    // LREAL
    IF UDINT_TO_INT(Expected.TypeClass) = IBaseLibrary.TypeClass.TYPE_LREAL THEN
        MEMCPY(destAddr := ADR(lrealExpected), srcAddr := Expected.pValue, n := SIZEOF(LREAL));
        MEMCPY(destAddr := ADR(lrealActual), srcAddr := Actual.pValue, n := SIZEOF(LREAL));
        AssertEquals_LREAL(Expected := lrealExpected, Actual := lrealActual, Delta := 0.0, Message := Message);
        RETURN;
    END_IF

    // LTIME
    IF UDINT_TO_INT(Expected.TypeClass) = IBaseLibrary.TypeClass.TYPE_LTIME THEN
        MEMCPY(destAddr := ADR(ltimeExpected), srcAddr := Expected.pValue, n := SIZEOF(LTIME));
        MEMCPY(destAddr := ADR(ltimeActual), srcAddr := Actual.pValue, n := SIZEOF(LTIME));
        AssertEquals_LTIME(Expected := ltimeExpected, Actual := ltimeActual, Message := Message);
        RETURN;
    END_IF

    // LWORD
    IF UDINT_TO_INT(Expected.TypeClass) = IBaseLibrary.TypeClass.TYPE_LWORD THEN
        MEMCPY(destAddr := ADR(lwordExpected), srcAddr := Expected.pValue, n := SIZEOF(LWORD));
        MEMCPY(destAddr := ADR(lwordActual), srcAddr := Actual.pValue, n := SIZEOF(LWORD));
        AssertEquals_LWORD(Expected := lwordExpected, Actual := lwordActual, Message := Message);
        RETURN;
    END_IF

    // REAL
    IF UDINT_TO_INT(Expected.TypeClass) = IBaseLibrary.TypeClass.TYPE_REAL THEN
        MEMCPY(destAddr := ADR(realExpected), srcAddr := Expected.pValue, n := SIZEOF(REAL));
        MEMCPY(destAddr := ADR(realActual), srcAddr := Actual.pValue, n := SIZEOF(REAL));
        AssertEquals_REAL(Expected := realExpected, Actual := realActual, Delta := 0.0, Message := Message);
        RETURN;
    END_IF

    // SINT
    IF UDINT_TO_INT(Expected.TypeClass) = IBaseLibrary.TypeClass.TYPE_SINT THEN
        MEMCPY(destAddr := ADR(sintExpected), srcAddr := Expected.pValue, n := SIZEOF(SINT));
        MEMCPY(destAddr := ADR(sintActual), srcAddr := Actual.pValue, n := SIZEOF(SINT));
        AssertEquals_SINT(Expected := sintExpected, Actual := sintActual, Message := Message);
        RETURN;
    END_IF

    // STRING
    IF UDINT_TO_INT(Expected.TypeClass) = IBaseLibrary.TypeClass.TYPE_STRING THEN
        MEMCPY(destAddr := ADR(stringExpected), srcAddr := Expected.pValue, n := DINT_TO_UDINT(Expected.diSize));
        MEMCPY(destAddr := ADR(stringActual), srcAddr := Actual.pValue, n := DINT_TO_UDINT(Actual.diSize));
        AssertEquals_STRING(Expected := stringExpected, Actual := stringActual, Message := Message);
        RETURN;
    END_IF

    // WSTRING
    IF UDINT_TO_INT(Expected.TypeClass) = IBaseLibrary.TypeClass.TYPE_WSTRING THEN
        MEMCPY(destAddr := ADR(wstringExpected), srcAddr := Expected.pValue, n := DINT_TO_UDINT(Expected.diSize));
        MEMCPY(destAddr := ADR(wstringActual), srcAddr := Actual.pValue, n := DINT_TO_UDINT(Actual.diSize));
        AssertEquals_WSTRING(Expected := wstringExpected, Actual := wstringActual, Message := Message);
        RETURN;
    END_IF

    // TIME
    IF UDINT_TO_INT(Expected.TypeClass) = IBaseLibrary.TypeClass.TYPE_TIME THEN
        MEMCPY(destAddr := ADR(timeExpected), srcAddr := Expected.pValue, n := SIZEOF(TIME));
        MEMCPY(destAddr := ADR(timeActual), srcAddr := Actual.pValue, n := SIZEOF(TIME));
        AssertEquals_TIME(Expected := timeExpected, Actual := timeActual, Message := Message);
        RETURN;
    END_IF

    // TIME_OF_DAY
    IF UDINT_TO_INT(Expected.TypeClass) = IBaseLibrary.TypeClass.TYPE_TIMEOFDAY THEN
        MEMCPY(destAddr := ADR(timeOfDayExpected), srcAddr := Expected.pValue, n := SIZEOF(TIME_OF_DAY));
        MEMCPY(destAddr := ADR(timeOfDayActual), srcAddr := Actual.pValue, n := SIZEOF(TIME_OF_DAY));
        AssertEquals_TIME_OF_DAY(Expected := timeOfDayExpected, Actual := timeOfDayActual, Message := Message);
        RETURN;
    END_IF

    // UDINT
    IF UDINT_TO_INT(Expected.TypeClass) = IBaseLibrary.TypeClass.TYPE_UDINT THEN
        MEMCPY(destAddr := ADR(udintExpected), srcAddr := Expected.pValue, n := SIZEOF(UDINT));
        MEMCPY(destAddr := ADR(udintActual), srcAddr := Actual.pValue, n := SIZEOF(UDINT));
        AssertEquals_UDINT(Expected := udintExpected, Actual := udintActual, Message := Message);
        RETURN;
    END_IF

    // UINT
    IF UDINT_TO_INT(Expected.TypeClass) = IBaseLibrary.TypeClass.TYPE_UINT THEN
        MEMCPY(destAddr := ADR(uintExpected), srcAddr := Expected.pValue, n := SIZEOF(UINT));
        MEMCPY(destAddr := ADR(uintActual), srcAddr := Actual.pValue, n := SIZEOF(UINT));
        AssertEquals_UINT(Expected := uintExpected, Actual := uintActual, Message := Message);
        RETURN;
    END_IF

    // ULINT
    IF UDINT_TO_INT(Expected.TypeClass) = IBaseLibrary.TypeClass.TYPE_ULINT THEN
        MEMCPY(destAddr := ADR(ulintExpected), srcAddr := Expected.pValue, n := SIZEOF(ULINT));
        MEMCPY(destAddr := ADR(ulintActual), srcAddr := Actual.pValue, n := SIZEOF(ULINT));
        AssertEquals_ULINT(Expected := ulintExpected, Actual := ulintActual, Message := Message);
        RETURN;
    END_IF

    // USINT
    IF UDINT_TO_INT(Expected.TypeClass) = IBaseLibrary.TypeClass.TYPE_USINT THEN
        MEMCPY(destAddr := ADR(usintExpected), srcAddr := Expected.pValue, n := SIZEOF(USINT));
        MEMCPY(destAddr := ADR(usintActual), srcAddr := Actual.pValue, n := SIZEOF(USINT));
        AssertEquals_USINT(Expected := usintExpected, Actual := usintActual, Message := Message);
        RETURN;
    END_IF

    // WORD
    IF UDINT_TO_INT(Expected.TypeClass) = IBaseLibrary.TypeClass.TYPE_WORD THEN
        MEMCPY(destAddr := ADR(wordExpected), srcAddr := Expected.pValue, n := SIZEOF(WORD));
        MEMCPY(destAddr := ADR(wordActual), srcAddr := Actual.pValue, n := SIZEOF(WORD));
        AssertEquals_WORD(Expected := wordExpected, Actual := wordActual, Message := Message);
        RETURN;
    END_IF

END_IF

(* If we've come to this row, it means that the data input is not any of the standard primitive data types, and thus
   we need to do special handling *)
TestInstancePath := AddTestNameToInstancePath(TestInstancePath := FindTestSuiteInstancePath());

IF DataTypesNotEquals THEN
    ExpectedDataString := CONCAT(STR1 := '(Type class = ', STR2 := F_AnyTypeClassToString((Expected.TypeClass)));
    ExpectedDataString := CONCAT(STR1 := ExpectedDataString, STR2 := ')');
    ActualDataString := CONCAT(STR1 := '(Type class = ', STR2 := F_AnyTypeClassToString(Actual.TypeClass));
    ActualDataString := CONCAT(STR1 := ActualDataString, STR2 := ')');
ELSIF DataSizeNotEquals THEN
    (* Take special care of STRING and WSTRING, as these can be declared with different sizes,
       although their content might be the same *)
    IF UDINT_TO_INT(Expected.TypeClass) = IBaseLibrary.TypeClass.TYPE_STRING THEN
        MEMCPY(destAddr := ADR(stringExpected), srcAddr := Expected.pValue, n := DINT_TO_UDINT(Expected.diSize));
        MEMCPY(destAddr := ADR(stringActual), srcAddr := Actual.pValue, n := DINT_TO_UDINT(Actual.diSize));
        ExpectedDataString := CONCAT(STR1 := '(Data size (LEN) = ', STR2 := INT_TO_STRING(LEN(STR := stringExpected)));
        ActualDataString := CONCAT(STR1 := '(Data size (LEN) = ', STR2 := INT_TO_STRING(LEN(STR := stringActual)));
    ELSIF UDINT_TO_INT(Expected.TypeClass) = IBaseLibrary.TypeClass.TYPE_WSTRING THEN
        MEMCPY(destAddr := ADR(wstringExpected), srcAddr := Expected.pValue, n := DINT_TO_UDINT(Expected.diSize));
        MEMCPY(destAddr := ADR(wstringActual), srcAddr := Actual.pValue, n := DINT_TO_UDINT(Actual.diSize));
        ExpectedDataString := CONCAT(STR1 := '(Data size (WLEN) = ', STR2 := INT_TO_STRING(WLEN(STR := wstringExpected)));
        ActualDataString := CONCAT(STR1 := '(Data size (WLEN) = ', STR2 := INT_TO_STRING(WLEN(STR := wstringActual)));
    ELSE
        ExpectedDataString := CONCAT(STR1 := '(Data size = ', STR2 := DINT_TO_STRING(Expected.diSize));
        ActualDataString := CONCAT(STR1 := '(Data size = ', STR2 := DINT_TO_STRING(Actual.diSize));
    END_IF
    ExpectedDataString := CONCAT(STR1 := ExpectedDataString, STR2 := ')');
    ActualDataString := CONCAT(STR1 := ActualDataString, STR2 := ')');
ELSIF DataContentNotEquals THEN
    FOR Count := 0 TO MIN(Expected.diSize-1, 38) BY 1 DO // One byte will equal two characters (example: 255 = 0xff, 1 = 0x01)
        ExpectedDataString := CONCAT(STR1 := ExpectedDataString,
                                                  STR2 := BYTE_TO_HEXSTR(in := Expected.pValue[Count],
                                                                                       iPrecision := 2,
                                                                                       bLoCase := FALSE));
    END_FOR
    ExpectedDataString := CONCAT(STR1 := '0x', STR2 := ExpectedDataString);

    FOR Count := 0 TO MIN(Actual.diSize-1, 38) BY 1 DO // One byte will equal two characters (example: 255 = 0xff, 1 = 0x01)
        ActualDataString := CONCAT(STR1 := ActualDataString,
                                                STR2 := BYTE_TO_HEXSTR(in := Actual.pValue[Count],
                                                                                     iPrecision := 2,
                                                                                     bLoCase := FALSE));
    END_FOR
    ActualDataString := CONCAT(STR1 := '0x', STR2 := ActualDataString);
END_IF

AssertResults.ReportResult(ExpectedSize := DINT_TO_UDINT(Expected.diSize),
                           ExpectedTypeClass := UDINT_TO_INT(Expected.TypeClass),
                           ExpectedValue := Expected.pValue,
                           ActualSize := DINT_TO_UDINT(Actual.diSize),
                           ActualTypeClass := UDINT_TO_INT(Actual.TypeClass),
                           ActualValue := Actual.pValue,
                           Message := Message,
                           TestInstancePath := TestInstancePath,
                           AlreadyReported => AlreadyReported);

IF NOT AlreadyReported AND (DataTypesNotEquals OR DataSizeNotEquals OR DataContentNotEquals) THEN
    SetTestFailed(AssertionType := E_AssertionType.Type_ANY,
                  AssertionMessage := Message);

    AssertMessageFormatter.LogAssertFailure(Expected := ExpectedDataString,
                                            Actual := ActualDataString,
                                            Message := Message,
                                            TestInstancePath := TestInstancePath);
END_IF
END_METHOD

// Asserts that two BOOLs are equal. If they are not, an assertion error is created.
METHOD PUBLIC AssertEquals_BOOL
VAR_INPUT
    Expected : BOOL; // BOOL expected value
    Actual : BOOL; // BOOL actual value
    Message : T_MaxString; // The identifying message for the assertion error
END_VAR
VAR
    AlreadyReported : BOOL;
    TestInstancePath : T_MaxString;
END_VAR
IF GVL_TcUnit.IgnoreCurrentTest OR GVL_TcUnit.CurrentTestIsFinished THEN
    RETURN;
END_IF

TestInstancePath := AddTestNameToInstancePath(TestInstancePath := FindTestSuiteInstancePath());

AssertResults.ReportResult(ExpectedSize := SIZEOF(Expected),
                           ExpectedTypeClass := IBaseLibrary.TypeClass.TYPE_BOOL,
                           ExpectedValue := ADR(Expected),
                           ActualSize := SIZEOF(Actual),
                           ActualTypeClass := IBaseLibrary.TypeClass.TYPE_BOOL,
                           ActualValue := ADR(Actual),
                           Message := Message,
                           TestInstancePath := TestInstancePath,
                           AlreadyReported => AlreadyReported);

IF NOT AlreadyReported AND Expected <> Actual THEN
    SetTestFailed(AssertionType := E_AssertionType.Type_BOOL,
                  AssertionMessage := Message);

    AssertMessageFormatter.LogAssertFailure(Expected := BOOL_TO_STRING(Expected),
                                            Actual := BOOL_TO_STRING(Actual),
                                            Message := Message,
                                            TestInstancePath := TestInstancePath);
END_IF
END_METHOD

// Asserts that two BYTEs are equal. If they are not, an assertion error is created.
METHOD PUBLIC AssertEquals_BYTE
VAR_INPUT
    Expected : BYTE; // BYTE expected value
    Actual : BYTE; // BYTE actual value
    Message : T_MaxString; // The identifying message for the assertion error
END_VAR
VAR
    TestInstancePath : T_MaxString;
    AlreadyReported : BOOL;
END_VAR
IF GVL_TcUnit.IgnoreCurrentTest OR GVL_TcUnit.CurrentTestIsFinished THEN
    RETURN;
END_IF

TestInstancePath := AddTestNameToInstancePath(TestInstancePath := FindTestSuiteInstancePath());

AssertResults.ReportResult(ExpectedSize := SIZEOF(Expected),
                           ExpectedTypeClass := IBaseLibrary.TypeClass.TYPE_BYTE,
                           ExpectedValue := ADR(Expected),
                           ActualSize := SIZEOF(Actual),
                           ActualTypeClass := IBaseLibrary.TypeClass.TYPE_BYTE,
                           ActualValue := ADR(Actual),
                           Message := Message,
                           TestInstancePath := TestInstancePath,
                           AlreadyReported => AlreadyReported);

IF NOT AlreadyReported AND Expected <> Actual THEN
    SetTestFailed(AssertionType := E_AssertionType.Type_BYTE,
                  AssertionMessage := Message);

    AssertMessageFormatter.LogAssertFailure(Expected := CONCAT(
                                                       STR1 := '0x',
                                                       STR2 := BYTE_TO_HEXSTR(in := Expected,
                                                                                            iPrecision := 2,
                                                                                            bLoCase := FALSE)),
                                            Actual := CONCAT(
                                                       STR1 := '0x',
                                                       STR2 := BYTE_TO_HEXSTR(in := Actual,
                                                                                            iPrecision := 2,
                                                                                            bLoCase := FALSE)),
                                            Message := Message,
                                            TestInstancePath := TestInstancePath);
END_IF
END_METHOD

// Asserts that two DATEs are equal. If they are not, an assertion error is created.
METHOD PUBLIC AssertEquals_DATE
VAR_INPUT
    Expected : DATE; // DATE expected value
    Actual : DATE; // DATE actual value
    Message : T_MaxString; // The identifying message for the assertion error
END_VAR
VAR
    TestInstancePath : T_MaxString;
    AlreadyReported : BOOL;
END_VAR
IF GVL_TcUnit.IgnoreCurrentTest OR GVL_TcUnit.CurrentTestIsFinished THEN
    RETURN;
END_IF

TestInstancePath := AddTestNameToInstancePath(TestInstancePath := FindTestSuiteInstancePath());

AssertResults.ReportResult(ExpectedSize := SIZEOF(Expected),
                           ExpectedTypeClass := IBaseLibrary.TypeClass.TYPE_DATE,
                           ExpectedValue := ADR(Expected),
                           ActualSize := SIZEOF(Actual),
                           ActualTypeClass := IBaseLibrary.TypeClass.TYPE_DATE,
                           ActualValue := ADR(Actual),
                           Message := Message,
                           TestInstancePath := TestInstancePath,
                           AlreadyReported => AlreadyReported);

IF NOT AlreadyReported AND Expected <> Actual THEN
    SetTestFailed(AssertionType := E_AssertionType.Type_DATE,
                  AssertionMessage := Message);

    AssertMessageFormatter.LogAssertFailure(Expected := DATE_TO_STRING(Expected),
                                            Actual := DATE_TO_STRING(Actual),
                                            Message := Message,
                                            TestInstancePath := TestInstancePath);
END_IF
END_METHOD

// Asserts that two DATE_AND_TIMEs are equal. If they are not, an assertion error is created.
METHOD PUBLIC AssertEquals_DATE_AND_TIME
VAR_INPUT
    Expected : DATE_AND_TIME; // DATE_AND_TIME expected value
    Actual : DATE_AND_TIME; // DATE_AND_TIME actual value
    Message : T_MaxString; // The identifying message for the assertion error
END_VAR
VAR
    TestInstancePath : T_MaxString;
    AlreadyReported : BOOL;
END_VAR
IF GVL_TcUnit.IgnoreCurrentTest OR GVL_TcUnit.CurrentTestIsFinished THEN
    RETURN;
END_IF

TestInstancePath := AddTestNameToInstancePath(TestInstancePath := FindTestSuiteInstancePath());

AssertResults.ReportResult(ExpectedSize := SIZEOF(Expected),
                           ExpectedTypeClass := IBaseLibrary.TypeClass.TYPE_DATEANDTIME,
                           ExpectedValue := ADR(Expected),
                           ActualSize := SIZEOF(Actual),
                           ActualTypeClass := IBaseLibrary.TypeClass.TYPE_DATEANDTIME,
                           ActualValue := ADR(Actual),
                           Message := Message,
                           TestInstancePath := TestInstancePath,
                           AlreadyReported => AlreadyReported);

IF NOT AlreadyReported AND Expected <> Actual THEN
    SetTestFailed(AssertionType := E_AssertionType.Type_DATE_AND_TIME,
                  AssertionMessage := Message);

    AssertMessageFormatter.LogAssertFailure(Expected := DT_TO_STRING(Expected),
                                            Actual := DT_TO_STRING(Actual),
                                            Message := Message,
                                            TestInstancePath := TestInstancePath);
END_IF
END_METHOD

// Asserts that two DINTs are equal. If they are not, an assertion error is created.
METHOD PUBLIC AssertEquals_DINT
VAR_INPUT
    Expected : DINT; // DINT expected value
    Actual : DINT; // DINT actual value
    Message : T_MaxString; // The identifying message for the assertion error
END_VAR
VAR
    TestInstancePath : T_MaxString;
    AlreadyReported : BOOL;
END_VAR
IF GVL_TcUnit.IgnoreCurrentTest OR GVL_TcUnit.CurrentTestIsFinished THEN
    RETURN;
END_IF

TestInstancePath := AddTestNameToInstancePath(TestInstancePath := FindTestSuiteInstancePath());

AssertResults.ReportResult(ExpectedSize := SIZEOF(Expected),
                           ExpectedTypeClass := IBaseLibrary.TypeClass.TYPE_DINT,
                           ExpectedValue := ADR(Expected),
                           ActualSize := SIZEOF(Actual),
                           ActualTypeClass := IBaseLibrary.TypeClass.TYPE_DINT,
                           ActualValue := ADR(Actual),
                           Message := Message,
                           TestInstancePath := TestInstancePath,
                           AlreadyReported => AlreadyReported);

IF NOT AlreadyReported AND Expected <> Actual THEN
    SetTestFailed(AssertionType := E_AssertionType.Type_DINT,
                  AssertionMessage := Message);

    AssertMessageFormatter.LogAssertFailure(Expected := DINT_TO_STRING(Expected),
                                            Actual := DINT_TO_STRING(Actual),
                                            Message := Message,
                                            TestInstancePath := TestInstancePath);
END_IF
END_METHOD

// Asserts that two DWORDs are equal. If they are not, an assertion error is created.
METHOD PUBLIC AssertEquals_DWORD
VAR_INPUT
    Expected : DWORD; // DWORD expected value
    Actual : DWORD; // DWORD actual value
    Message : T_MaxString; // The identifying message for the assertion error
END_VAR
VAR
    TestInstancePath : T_MaxString;
    AlreadyReported : BOOL;
END_VAR
IF GVL_TcUnit.IgnoreCurrentTest OR GVL_TcUnit.CurrentTestIsFinished THEN
    RETURN;
END_IF

TestInstancePath := AddTestNameToInstancePath(TestInstancePath := FindTestSuiteInstancePath());

AssertResults.ReportResult(ExpectedSize := SIZEOF(Expected),
                           ExpectedTypeClass := IBaseLibrary.TypeClass.TYPE_DWORD,
                           ExpectedValue := ADR(Expected),
                           ActualSize := SIZEOF(Actual),
                           ActualTypeClass := IBaseLibrary.TypeClass.TYPE_DWORD,
                           ActualValue := ADR(Actual),
                           Message := Message,
                           TestInstancePath := TestInstancePath,
                           AlreadyReported => AlreadyReported);

IF NOT AlreadyReported AND Expected <> Actual THEN
    SetTestFailed(AssertionType := E_AssertionType.Type_DWORD,
                  AssertionMessage := Message);

    AssertMessageFormatter.LogAssertFailure(Expected := CONCAT(
                                                            STR1 := '0x',
                                                            STR2 := DWORD_TO_HEXSTR(in := Expected,
                                                                                                  iPrecision := 8,
                                                                                                  bLoCase := FALSE)),
                                            Actual := CONCAT(
                                                           STR1 := '0x',
                                                           STR2 := DWORD_TO_HEXSTR(in := Actual,
                                                                                                 iPrecision := 8,
                                                                                                 bLoCase := FALSE)),
                                            Message := Message,
                                            TestInstancePath := TestInstancePath);
END_IF
END_METHOD

// Asserts that two INTs are equal. If they are not, an assertion error is created.
METHOD PUBLIC AssertEquals_INT
VAR_INPUT
    Expected : INT; // INT expected value
    Actual : INT; // INT actual value
    Message : T_MaxString; // The identifying message for the assertion error
END_VAR
VAR
    TestInstancePath : T_MaxString;
    AlreadyReported : BOOL;
END_VAR
IF GVL_TcUnit.IgnoreCurrentTest OR GVL_TcUnit.CurrentTestIsFinished THEN
    RETURN;
END_IF

TestInstancePath := AddTestNameToInstancePath(TestInstancePath := FindTestSuiteInstancePath());

AssertResults.ReportResult(ExpectedSize := SIZEOF(Expected),
                           ExpectedTypeClass := IBaseLibrary.TypeClass.TYPE_INT,
                           ExpectedValue := ADR(Expected),
                           ActualSize := SIZEOF(Actual),
                           ActualTypeClass := IBaseLibrary.TypeClass.TYPE_INT,
                           ActualValue := ADR(Actual),
                           Message := Message,
                           TestInstancePath := TestInstancePath,
                           AlreadyReported => AlreadyReported);

IF NOT AlreadyReported AND Expected <> Actual THEN
    SetTestFailed(AssertionType := E_AssertionType.Type_INT,
                  AssertionMessage := Message);

    AssertMessageFormatter.LogAssertFailure(Expected := INT_TO_STRING(Expected),
                                            Actual := INT_TO_STRING(Actual),
                                            Message := Message,
                                            TestInstancePath := TestInstancePath);
END_IF
END_METHOD

// Asserts that two LINTs are equal. If they are not, an assertion error is created.
METHOD PUBLIC AssertEquals_LINT
VAR_INPUT
    Expected : LINT; // LINT expected value
    Actual : LINT; // LINT actual value
    Message : T_MaxString; // The identifying message for the assertion error
END_VAR
VAR
    TestInstancePath : T_MaxString;
    AlreadyReported : BOOL;
END_VAR
IF GVL_TcUnit.IgnoreCurrentTest OR GVL_TcUnit.CurrentTestIsFinished THEN
    RETURN;
END_IF

TestInstancePath := AddTestNameToInstancePath(TestInstancePath := FindTestSuiteInstancePath());

AssertResults.ReportResult(ExpectedSize := SIZEOF(Expected),
                           ExpectedTypeClass := IBaseLibrary.TypeClass.TYPE_LINT,
                           ExpectedValue := ADR(Expected),
                           ActualSize := SIZEOF(Actual),
                           ActualTypeClass := IBaseLibrary.TypeClass.TYPE_LINT,
                           ActualValue := ADR(Actual),
                           Message := Message,
                           TestInstancePath := TestInstancePath,
                           AlreadyReported => AlreadyReported);

IF NOT AlreadyReported AND Expected <> Actual THEN
    SetTestFailed(AssertionType := E_AssertionType.Type_LINT,
                  AssertionMessage := Message);

    AssertMessageFormatter.LogAssertFailure(Expected := LINT_TO_STRING(Expected),
                                            Actual := LINT_TO_STRING(Actual),
                                            Message := Message,
                                            TestInstancePath := TestInstancePath);
END_IF
END_METHOD

// Asserts that two LREALs are equal to within a positive delta. If they are not, an assertion error is created.
METHOD PUBLIC AssertEquals_LREAL
VAR_INPUT
    Expected : LREAL; // LREAL expected value
    Actual : LREAL; // LREAL actual value
    Delta : LREAL; // The maximum delta between the absolute value of expected and actual for which both numbers are still considered equal
    Message : T_MaxString; // The identifying message for the assertion error
END_VAR
VAR
    TestInstancePath : T_MaxString;
    AlreadyReported : BOOL;
END_VAR
IF GVL_TcUnit.IgnoreCurrentTest OR GVL_TcUnit.CurrentTestIsFinished THEN
    RETURN;
END_IF

TestInstancePath := AddTestNameToInstancePath(TestInstancePath := FindTestSuiteInstancePath());

AssertResults.ReportResult(ExpectedSize := SIZEOF(Expected),
                           ExpectedTypeClass := IBaseLibrary.TypeClass.TYPE_LREAL,
                           ExpectedValue := ADR(Expected),
                           ActualSize := SIZEOF(Actual),
                           ActualTypeClass := IBaseLibrary.TypeClass.TYPE_LREAL,
                           ActualValue := ADR(Actual),
                           Message := Message,
                           TestInstancePath := TestInstancePath,
                           AlreadyReported => AlreadyReported);

IF NOT AlreadyReported AND ABS(Expected - Actual) > Delta THEN
    SetTestFailed(AssertionType := E_AssertionType.Type_LREAL,
                  AssertionMessage := Message);

    AssertMessageFormatter.LogAssertFailure(Expected := LREAL_TO_STRING(Expected),
                                            Actual := LREAL_TO_STRING(Actual),
                                            Message := Message,
                                            TestInstancePath := TestInstancePath);
END_IF
END_METHOD

// Asserts that two LTIMEs are equal. If they are not, an assertion error is created.
METHOD PUBLIC AssertEquals_LTIME
VAR_INPUT
    Expected : LTIME; // LTIME expected value
    Actual : LTIME; // LTIME actual value
    Message : T_MaxString; // The identifying message for the assertion error
END_VAR
VAR
    TestInstancePath : T_MaxString;
    AlreadyReported : BOOL;
END_VAR
IF GVL_TcUnit.IgnoreCurrentTest OR GVL_TcUnit.CurrentTestIsFinished THEN
    RETURN;
END_IF

TestInstancePath := AddTestNameToInstancePath(TestInstancePath := FindTestSuiteInstancePath());

AssertResults.ReportResult(ExpectedSize := SIZEOF(Expected),
                           ExpectedTypeClass := IBaseLibrary.TypeClass.TYPE_LTIME,
                           ExpectedValue := ADR(Expected),
                           ActualSize := SIZEOF(Actual),
                           ActualTypeClass := IBaseLibrary.TypeClass.TYPE_LTIME,
                           ActualValue := ADR(Actual),
                           Message := Message,
                           TestInstancePath := TestInstancePath,
                           AlreadyReported => AlreadyReported);

IF NOT AlreadyReported AND Expected <> Actual THEN
    SetTestFailed(AssertionType := E_AssertionType.Type_LTIME,
                  AssertionMessage := Message);

    AssertMessageFormatter.LogAssertFailure(Expected := LTIME_TO_STRING(Expected),
                                            Actual := LTIME_TO_STRING(Actual),
                                            Message := Message,
                                            TestInstancePath := TestInstancePath);
END_IF
END_METHOD

// Asserts that two LWORDs are equal. If they are not, an assertion error is created.
METHOD PUBLIC AssertEquals_LWORD
VAR_INPUT
    Expected : LWORD; // LWORD expected value
    Actual : LWORD; // LWORD actual value
    Message : T_MaxString; // The identifying message for the assertion error
END_VAR
VAR
    TestInstancePath : T_MaxString;
    AlreadyReported : BOOL;
END_VAR
IF GVL_TcUnit.IgnoreCurrentTest OR GVL_TcUnit.CurrentTestIsFinished THEN
    RETURN;
END_IF

TestInstancePath := AddTestNameToInstancePath(TestInstancePath := FindTestSuiteInstancePath());

AssertResults.ReportResult(ExpectedSize := SIZEOF(Expected),
                           ExpectedTypeClass := IBaseLibrary.TypeClass.TYPE_LWORD,
                           ExpectedValue := ADR(Expected),
                           ActualSize := SIZEOF(Actual),
                           ActualTypeClass := IBaseLibrary.TypeClass.TYPE_LWORD,
                           ActualValue := ADR(Actual),
                           Message := Message,
                           TestInstancePath := TestInstancePath,
                           AlreadyReported => AlreadyReported);

IF NOT AlreadyReported AND Expected <> Actual THEN
    SetTestFailed(AssertionType := E_AssertionType.Type_LWORD,
                  AssertionMessage := Message);

    AssertMessageFormatter.LogAssertFailure(Expected := CONCAT(
                                                            STR1 := '0x',
                                                            STR2 := LWORD_TO_HEXSTR(in := Expected,
                                                                                                  iPrecision := 16,
                                                                                                  bLoCase := FALSE)),
                                            Actual := CONCAT(
                                                            STR1 := '0x',
                                                            STR2 := LWORD_TO_HEXSTR(in := Actual,
                                                                                                  iPrecision := 16,
                                                                                                  bLoCase := FALSE)),
                                            Message := Message,
                                            TestInstancePath := TestInstancePath);
END_IF
END_METHOD

// Asserts that two REALs are equal to within a positive delta. If they are not, an assertion error is created.
METHOD PUBLIC AssertEquals_REAL
VAR_INPUT
    Expected : REAL; // REAL expected value
    Actual : REAL; // REAL actual value
    Delta : REAL;  // The maximum delta between the absolute value of expected and actual for which both numbers are still considered equal
    Message : T_MaxString; // The identifying message for the assertion error
END_VAR
VAR
    TestInstancePath : T_MaxString;
    AlreadyReported : BOOL;
END_VAR
IF GVL_TcUnit.IgnoreCurrentTest OR GVL_TcUnit.CurrentTestIsFinished THEN
    RETURN;
END_IF

TestInstancePath := AddTestNameToInstancePath(TestInstancePath := FindTestSuiteInstancePath());

AssertResults.ReportResult(ExpectedSize := SIZEOF(Expected),
                           ExpectedTypeClass := IBaseLibrary.TypeClass.TYPE_REAL,
                           ExpectedValue := ADR(Expected),
                           ActualSize := SIZEOF(Actual),
                           ActualTypeClass := IBaseLibrary.TypeClass.TYPE_REAL,
                           ActualValue := ADR(Actual),
                           Message := Message,
                           TestInstancePath := TestInstancePath,
                           AlreadyReported => AlreadyReported);

IF NOT AlreadyReported AND ABS(Expected - Actual) > Delta THEN
    SetTestFailed(AssertionType := E_AssertionType.Type_REAL,
                  AssertionMessage := Message);

    AssertMessageFormatter.LogAssertFailure(Expected := REAL_TO_STRING(Expected),
                                            Actual := REAL_TO_STRING(Actual),
                                            Message := Message,
                                            TestInstancePath := TestInstancePath);
END_IF
END_METHOD

// Asserts that two SINTs are equal. If they are not, an assertion error is created.
METHOD PUBLIC AssertEquals_SINT
VAR_INPUT
    Expected : SINT; // SINT expected value
    Actual : SINT; // SINT actual value
    Message : T_MaxString; // The identifying message for the assertion error
END_VAR
VAR
    TestInstancePath : T_MaxString;
    AlreadyReported : BOOL;
END_VAR
IF GVL_TcUnit.IgnoreCurrentTest OR GVL_TcUnit.CurrentTestIsFinished THEN
    RETURN;
END_IF

TestInstancePath := AddTestNameToInstancePath(TestInstancePath := FindTestSuiteInstancePath());

AssertResults.ReportResult(ExpectedSize := SIZEOF(Expected),
                           ExpectedTypeClass := IBaseLibrary.TypeClass.TYPE_SINT,
                           ExpectedValue := ADR(Expected),
                           ActualSize := SIZEOF(Actual),
                           ActualTypeClass := IBaseLibrary.TypeClass.TYPE_SINT,
                           ActualValue := ADR(Actual),
                           Message := Message,
                           TestInstancePath := TestInstancePath,
                           AlreadyReported => AlreadyReported);

IF NOT AlreadyReported AND Expected <> Actual THEN
    SetTestFailed(AssertionType := E_AssertionType.Type_SINT,
                  AssertionMessage := Message);

    AssertMessageFormatter.LogAssertFailure(Expected := SINT_TO_STRING(Expected),
                                            Actual := SINT_TO_STRING(Actual),
                                            Message := Message,
                                            TestInstancePath := TestInstancePath);
END_IF
END_METHOD

// Asserts that two STRINGs are equal. If they are not, an assertion error is created.
METHOD PUBLIC AssertEquals_STRING
VAR_INPUT
    Expected : T_MaxString; // STRING expected value
    Actual : T_MaxString; // STRING actual value
    Message : T_MaxString; // The identifying message for the assertion error
END_VAR
VAR
    TestInstancePath : T_MaxString;
    AlreadyReported : BOOL;
END_VAR
IF GVL_TcUnit.IgnoreCurrentTest OR GVL_TcUnit.CurrentTestIsFinished THEN
    RETURN;
END_IF

TestInstancePath := AddTestNameToInstancePath(TestInstancePath := FindTestSuiteInstancePath());

AssertResults.ReportResult(ExpectedSize := SIZEOF(Expected),
                           ExpectedTypeClass := IBaseLibrary.TypeClass.TYPE_STRING,
                           ExpectedValue := ADR(Expected),
                           ActualSize := SIZEOF(Actual),
                           ActualTypeClass := IBaseLibrary.TypeClass.TYPE_STRING,
                           ActualValue := ADR(Actual),
                           Message := Message,
                           TestInstancePath := TestInstancePath,
                           AlreadyReported => AlreadyReported);

IF NOT AlreadyReported AND (LEN(STR := Expected) <> LEN(STR := Actual) OR (Expected <> Actual)) THEN
    SetTestFailed(AssertionType := E_AssertionType.Type_STRING,
                  AssertionMessage := Message);

    AssertMessageFormatter.LogAssertFailure(Expected := Expected,
                                            Actual := Actual,
                                            Message := Message,
                                            TestInstancePath := TestInstancePath);
END_IF
END_METHOD

// Asserts that two TIMEs are equal. If they are not, an assertion error is created.
METHOD PUBLIC AssertEquals_TIME
VAR_INPUT
    Expected : TIME; // TIME expected value
    Actual : TIME; // TIME actual value
    Message : T_MaxString; // The identifying message for the assertion error
END_VAR
VAR
    TestInstancePath : T_MaxString;
    AlreadyReported : BOOL;
END_VAR
IF GVL_TcUnit.IgnoreCurrentTest OR GVL_TcUnit.CurrentTestIsFinished THEN
    RETURN;
END_IF

TestInstancePath := AddTestNameToInstancePath(TestInstancePath := FindTestSuiteInstancePath());

AssertResults.ReportResult(ExpectedSize := SIZEOF(Expected),
                           ExpectedTypeClass := IBaseLibrary.TypeClass.TYPE_TIME,
                           ExpectedValue := ADR(Expected),
                           ActualSize := SIZEOF(Actual),
                           ActualTypeClass := IBaseLibrary.TypeClass.TYPE_TIME,
                           ActualValue := ADR(Actual),
                           Message := Message,
                           TestInstancePath := TestInstancePath,
                           AlreadyReported => AlreadyReported);

IF NOT AlreadyReported AND Expected <> Actual THEN
    SetTestFailed(AssertionType := E_AssertionType.Type_TIME,
                  AssertionMessage := Message);

    AssertMessageFormatter.LogAssertFailure(Expected := TIME_TO_STRING(Expected),
                                            Actual := TIME_TO_STRING(Actual),
                                            Message := Message,
                                            TestInstancePath := TestInstancePath);
END_IF
END_METHOD

// Asserts that two TIME_OF_DAYs are equal. If they are not, an assertion error is created.
METHOD PUBLIC AssertEquals_TIME_OF_DAY
VAR_INPUT
    Expected : TIME_OF_DAY; // TIME_OF_DAY expected value
    Actual : TIME_OF_DAY; // TIME_OF_DAY actual value
    Message : T_MaxString; // The identifying message for the assertion error
END_VAR
VAR
    TestInstancePath : T_MaxString;
    AlreadyReported : BOOL;
END_VAR
IF GVL_TcUnit.IgnoreCurrentTest OR GVL_TcUnit.CurrentTestIsFinished THEN
    RETURN;
END_IF

TestInstancePath := AddTestNameToInstancePath(TestInstancePath := FindTestSuiteInstancePath());

AssertResults.ReportResult(ExpectedSize := SIZEOF(Expected),
                           ExpectedTypeClass := IBaseLibrary.TypeClass.TYPE_TIMEOFDAY,
                           ExpectedValue := ADR(Expected),
                           ActualSize := SIZEOF(Actual),
                           ActualTypeClass := IBaseLibrary.TypeClass.TYPE_TIMEOFDAY,
                           ActualValue := ADR(Actual),
                           Message := Message,
                           TestInstancePath := TestInstancePath,
                           AlreadyReported => AlreadyReported);

IF NOT AlreadyReported AND Expected <> Actual THEN
    SetTestFailed(AssertionType := E_AssertionType.Type_TIME_OF_DAY,
                  AssertionMessage := Message);

    AssertMessageFormatter.LogAssertFailure(Expected := TOD_TO_STRING(Expected),
                                            Actual := TOD_TO_STRING(Actual),
                                            Message := Message,
                                            TestInstancePath := TestInstancePath);
END_IF
END_METHOD

// Asserts that two UDINTs are equal. If they are not, an assertion error is created.
METHOD PUBLIC AssertEquals_UDINT
VAR_INPUT
    Expected : UDINT; // UDINT expected value
    Actual : UDINT; // UDINT actual value
    Message : T_MaxString; // The identifying message for the assertion error
END_VAR
VAR
    TestInstancePath : T_MaxString;
    AlreadyReported : BOOL;
END_VAR
IF GVL_TcUnit.IgnoreCurrentTest OR GVL_TcUnit.CurrentTestIsFinished THEN
    RETURN;
END_IF

TestInstancePath := AddTestNameToInstancePath(TestInstancePath := FindTestSuiteInstancePath());

AssertResults.ReportResult(ExpectedSize := SIZEOF(Expected),
                           ExpectedTypeClass := IBaseLibrary.TypeClass.TYPE_UDINT,
                           ExpectedValue := ADR(Expected),
                           ActualSize := SIZEOF(Actual),
                           ActualTypeClass := IBaseLibrary.TypeClass.TYPE_UDINT,
                           ActualValue := ADR(Actual),
                           Message := Message,
                           TestInstancePath := TestInstancePath,
                           AlreadyReported => AlreadyReported);

IF NOT AlreadyReported AND Expected <> Actual THEN
    SetTestFailed(AssertionType := E_AssertionType.Type_UDINT,
                  AssertionMessage := Message);

    AssertMessageFormatter.LogAssertFailure(Expected := UDINT_TO_STRING(Expected),
                                            Actual := UDINT_TO_STRING(Actual),
                                            Message := Message,
                                            TestInstancePath := TestInstancePath);
END_IF
END_METHOD

// Asserts that two UINTs are equal. If they are not, an assertion error is created.
METHOD PUBLIC AssertEquals_UINT
VAR_INPUT
    Expected : UINT; // UINT expected value
    Actual : UINT; // UINT actual value
    Message : T_MaxString; // The identifying message for the assertion error
END_VAR
VAR
    TestInstancePath : T_MaxString;
    AlreadyReported : BOOL;
END_VAR
IF GVL_TcUnit.IgnoreCurrentTest OR GVL_TcUnit.CurrentTestIsFinished THEN
    RETURN;
END_IF

TestInstancePath := AddTestNameToInstancePath(TestInstancePath := FindTestSuiteInstancePath());

AssertResults.ReportResult(ExpectedSize := SIZEOF(Expected),
                           ExpectedTypeClass := IBaseLibrary.TypeClass.TYPE_UINT,
                           ExpectedValue := ADR(Expected),
                           ActualSize := SIZEOF(Actual),
                           ActualTypeClass := IBaseLibrary.TypeClass.TYPE_UINT,
                           ActualValue := ADR(Actual),
                           Message := Message,
                           TestInstancePath := TestInstancePath,
                           AlreadyReported => AlreadyReported);

IF NOT AlreadyReported AND Expected <> Actual THEN
    SetTestFailed(AssertionType := E_AssertionType.Type_UINT,
                  AssertionMessage := Message);

    AssertMessageFormatter.LogAssertFailure(Expected := UINT_TO_STRING(Expected),
                                            Actual := UINT_TO_STRING(Actual),
                                            Message := Message,
                                            TestInstancePath := TestInstancePath);
END_IF
END_METHOD

// Asserts that two ULINTs are equal. If they are not, an assertion error is created.
METHOD PUBLIC AssertEquals_ULINT
VAR_INPUT
    Expected : ULINT; // ULINT expected value
    Actual : ULINT; // ULINT actual value
    Message : T_MaxString; // The identifying message for the assertion error
END_VAR
VAR
    TestInstancePath : T_MaxString;
    AlreadyReported : BOOL;
END_VAR
IF GVL_TcUnit.IgnoreCurrentTest OR GVL_TcUnit.CurrentTestIsFinished THEN
    RETURN;
END_IF

TestInstancePath := AddTestNameToInstancePath(TestInstancePath := FindTestSuiteInstancePath());

AssertResults.ReportResult(ExpectedSize := SIZEOF(Expected),
                           ExpectedTypeClass := IBaseLibrary.TypeClass.TYPE_ULINT,
                           ExpectedValue := ADR(Expected),
                           ActualSize := SIZEOF(Actual),
                           ActualTypeClass := IBaseLibrary.TypeClass.TYPE_ULINT,
                           ActualValue := ADR(Actual),
                           Message := Message,
                           TestInstancePath := TestInstancePath,
                           AlreadyReported => AlreadyReported);

IF NOT AlreadyReported AND Expected <> Actual THEN
    SetTestFailed(AssertionType := E_AssertionType.Type_ULINT,
                  AssertionMessage := Message);

    AssertMessageFormatter.LogAssertFailure(Expected := ULINT_TO_STRING(Expected),
                                            Actual := ULINT_TO_STRING(Actual),
                                            Message := Message,
                                            TestInstancePath := TestInstancePath);
END_IF
END_METHOD

// Asserts that two USINTs are equal. If they are not, an assertion error is created.
METHOD PUBLIC AssertEquals_USINT
VAR_INPUT
    Expected : USINT; // USINT expected value
    Actual : USINT; // USINT actual value
    Message : T_MaxString; // The identifying message for the assertion error
END_VAR
VAR
    AlreadyReported : BOOL;
    TestInstancePath : T_MaxString;
END_VAR
IF GVL_TcUnit.IgnoreCurrentTest OR GVL_TcUnit.CurrentTestIsFinished THEN
    RETURN;
END_IF

TestInstancePath := AddTestNameToInstancePath(TestInstancePath := FindTestSuiteInstancePath());

AssertResults.ReportResult(ExpectedSize := SIZEOF(Expected),
                           ExpectedTypeClass := IBaseLibrary.TypeClass.TYPE_USINT,
                           ExpectedValue := ADR(Expected),
                           ActualSize := SIZEOF(Actual),
                           ActualTypeClass := IBaseLibrary.TypeClass.TYPE_USINT,
                           ActualValue := ADR(Actual),
                           Message := Message,
                           TestInstancePath := TestInstancePath,
                           AlreadyReported => AlreadyReported);

IF NOT AlreadyReported AND Expected <> Actual THEN
    SetTestFailed(AssertionType := E_AssertionType.Type_USINT,
                  AssertionMessage := Message);

    AssertMessageFormatter.LogAssertFailure(Expected := USINT_TO_STRING(Expected),
                                            Actual := USINT_TO_STRING(Actual),
                                            Message := Message,
                                            TestInstancePath := TestInstancePath);
END_IF
END_METHOD

// Asserts that two WORDs are equal. If they are not, an assertion error is created.
METHOD PUBLIC AssertEquals_WORD
VAR_INPUT
    Expected : WORD; // WORD expected value
    Actual : WORD; // WORD actual value
    Message : T_MaxString; // The identifying message for the assertion error
END_VAR
VAR
    TestInstancePath : T_MaxString;
    AlreadyReported : BOOL;
END_VAR
IF GVL_TcUnit.IgnoreCurrentTest OR GVL_TcUnit.CurrentTestIsFinished THEN
    RETURN;
END_IF

TestInstancePath := AddTestNameToInstancePath(TestInstancePath := FindTestSuiteInstancePath());

AssertResults.ReportResult(ExpectedSize := SIZEOF(Expected),
                           ExpectedTypeClass := IBaseLibrary.TypeClass.TYPE_WORD,
                           ExpectedValue := ADR(Expected),
                           ActualSize := SIZEOF(Actual),
                           ActualTypeClass := IBaseLibrary.TypeClass.TYPE_WORD,
                           ActualValue := ADR(Actual),
                           Message := Message,
                           TestInstancePath := TestInstancePath,
                           AlreadyReported => AlreadyReported);

IF NOT AlreadyReported AND Expected <> Actual THEN
    SetTestFailed(AssertionType := E_AssertionType.Type_WORD,
                  AssertionMessage := Message);

    AssertMessageFormatter.LogAssertFailure(Expected := CONCAT(
                                                            STR1 := '0x',
                                                            STR2 := WORD_TO_HEXSTR(in := Expected,
                                                                                                 iPrecision := 4,
                                                                                                 bLoCase := FALSE)),
                                            Actual := CONCAT(
                                                            STR1 := '0x',
                                                            STR2 := WORD_TO_HEXSTR(in := Actual,
                                                                                                 iPrecision := 4,
                                                                                                 bLoCase := FALSE)),
                                            Message := Message,
                                            TestInstancePath := TestInstancePath);
END_IF
END_METHOD

// Asserts that two WSTRINGs are equal. If they are not, an assertion error is created.
METHOD PUBLIC AssertEquals_WSTRING
VAR_INPUT
    Expected : WSTRING(255); // WSTRING expected value
    Actual : WSTRING(255); // WSTRING actual value
    Message : T_MaxString; // The identifying message for the assertion error
END_VAR
VAR
    TestInstancePath : T_MaxString;
    AlreadyReported : BOOL;
END_VAR
IF GVL_TcUnit.IgnoreCurrentTest OR GVL_TcUnit.CurrentTestIsFinished THEN
    RETURN;
END_IF

TestInstancePath := AddTestNameToInstancePath(TestInstancePath := FindTestSuiteInstancePath());

AssertResults.ReportResult(ExpectedSize := SIZEOF(Expected),
                           ExpectedTypeClass := IBaseLibrary.TypeClass.TYPE_WSTRING,
                           ExpectedValue := ADR(Expected),
                           ActualSize := SIZEOF(Actual),
                           ActualTypeClass := IBaseLibrary.TypeClass.TYPE_WSTRING,
                           ActualValue := ADR(Actual),
                           Message := Message,
                           TestInstancePath := TestInstancePath,
                           AlreadyReported => AlreadyReported);

IF NOT AlreadyReported AND (WLEN(STR := Expected) <> WLEN(STR := Actual) OR (Expected <> Actual)) THEN
    SetTestFailed(AssertionType := E_AssertionType.Type_WSTRING,
                  AssertionMessage := Message);

    AssertMessageFormatter.LogAssertFailure(Expected := 'Not possible to print EXP unicode WSTRING value',
                                            Actual := 'Not possible to print ACT unicode WSTRING value',
                                            Message := Message,
                                            TestInstancePath := TestInstancePath);
END_IF
END_METHOD

// Asserts that a condition is false. If it is not, an assertion error is created.
METHOD PUBLIC AssertFalse
VAR_INPUT
    Condition : BOOL; // Condition to be checked
    Message : T_MaxString; // The identifying message for the assertion error
END_VAR
AssertEquals_BOOL(Expected := FALSE,
                  Actual := Condition,
                  Message := Message);
END_METHOD

// Asserts that a condition is true. If it is not, an assertion error is created.
METHOD PUBLIC AssertTrue
VAR_INPUT
    Condition : BOOL; // Condition to be checked
    Message : T_MaxString; // The identifying message for the assertion error
END_VAR
AssertEquals_BOOL(Expected := TRUE,
                  Actual := Condition,
                  Message := Message);
END_METHOD

METHOD INTERNAL CalculateAndSetNumberOfAssertsForTest
VAR_INPUT
    TestName : T_MaxString;
END_VAR
VAR
    TestInstancePath : T_MaxString;
    TotalNumberOfAsserts : UINT;
    NumberOfAsserts : UINT;
    NumberOfArrayAsserts : UINT;
    
    IteratorCounter : UINT;
END_VAR
TestInstancePath := AddTestNameToInstancePath(FindTestSuiteInstancePath());
NumberOfAsserts := AssertResults.GetNumberOfAssertsForTest(CompleteTestInstancePath := TestInstancePath);
NumberOfArrayAsserts := AssertArrayResults.GetNumberOfArrayAssertsForTest(CompleteTestInstancePath := TestInstancePath);
TotalNumberOfAsserts := NumberOfAsserts + NumberOfArrayAsserts;

IF TotalNumberOfAsserts > 0 THEN
    IF NumberOfTests > 0 THEN
        FOR IteratorCounter := 1 TO NumberOfTests BY 1 DO
            IF Tests[IteratorCounter].GetName() = TestName THEN
                Tests[IteratorCounter].SetNumberOfAssertions(NoOfAssertions := TotalNumberOfAsserts);
                RETURN;
            END_IF
        END_FOR
    END_IF
END_IF
END_METHOD

METHOD INTERNAL CalculateDuration
VAR_INPUT
    FinishedAt : LWORD; // CPU cycle counter with 100ns precision
END_VAR
IF Duration = 0.0 THEN
	Duration := LWORD_TO_LREAL(FinishedAt - StartedAt) * GVL_TcUnit.HundredNanosecondToSecond; // Seconds
	TraceWithSeverity(
		Message := CONCAT(CONCAT('SUITE COMPLETE: ', InstancePath),
				   CONCAT(' - ', CONCAT(UINT_TO_STRING(GetNumberOfSuccessfulTests()), CONCAT(' passed, ',
				   CONCAT(UINT_TO_STRING(GetNumberOfFailedTests()), CONCAT(' failed, ',
				   CONCAT(UINT_TO_STRING(GetNumberOfSkippedTests()), CONCAT(' skipped (',
				   CONCAT(LREAL_TO_STRING(Duration), 's)'))))))))),
		Severity := Global.TcEventSeverity.Info);
END_IF
END_METHOD

METHOD FB_init : BOOL
VAR_INPUT
    bInitRetains : BOOL; // if TRUE, the retain variables are initialized (warm start / cold start)
    bInCopyCode : BOOL;  // if TRUE, the instance afterwards gets moved into the copy code (online change)
END_VAR
GVL_TcUnit.NumberOfInitializedTestSuites := GVL_TcUnit.NumberOfInitializedTestSuites + 1;
GVL_TcUnit.TestSuiteAddresses[GVL_TcUnit.NumberOfInitializedTestSuites] := THIS;
END_METHOD

// Searches for the instance path of the calling function block
METHOD PRIVATE FindTestSuiteInstancePath : T_MaxString
FindTestSuiteInstancePath := GetInstancePath();
END_METHOD

METHOD INTERNAL GetDuration : LREAL
GetDuration := Duration;
END_METHOD

METHOD INTERNAL GetHasStartedRunning : BOOL
GetHasStartedRunning := StartedAt > 0;
END_METHOD

METHOD INTERNAL GetInstancePath : T_MaxString
GetInstancePath := InstancePath;
END_METHOD

METHOD INTERNAL GetNumberOfFailedTests : UINT
VAR
    Counter : UINT;
    FailedTestsCount : UINT;
    NumberOfTestsToAnalyse : UINT(1..GVL_Param_TcUnit.MaxNumberOfTestsForEachTestSuite);
    NumberOfTestOverArrayLimit : UINT;
END_VAR
// Limit the test analyse to the max array limit of 'Tests[]'
NumberOfTestsToAnalyse := GetNumberOfTestsToAnalyse();
IF GetNumberOfTests() > NumberOfTestsToAnalyse THEN
    NumberOfTestOverArrayLimit := GetNumberOfTests()-NumberOfTestsToAnalyse;
END_IF

FOR Counter := 1 TO NumberOfTestsToAnalyse BY 1 DO
    IF Tests[Counter].IsFailed() THEN
        FailedTestsCount := FailedTestsCount + 1;
    END_IF
END_FOR

GetNumberOfFailedTests := FailedTestsCount + NumberOfTestOverArrayLimit;
END_METHOD

METHOD INTERNAL GetNumberOfSkippedTests : UINT
VAR
    Counter : UINT;
    SkippedTestsCount : UINT;
    NumberOfTestsToAnalyse : UINT(1..GVL_Param_TcUnit.MaxNumberOfTestsForEachTestSuite);
END_VAR
// Limit the test analyse to the max array limit of 'Tests[]'
NumberOfTestsToAnalyse := GetNumberOfTestsToAnalyse();

FOR Counter := 1 TO NumberOfTestsToAnalyse BY 1 DO
    IF Tests[Counter].IsSkipped() THEN
        SkippedTestsCount := SkippedTestsCount + 1;
    END_IF
END_FOR

GetNumberOfSkippedTests := SkippedTestsCount;
END_METHOD

METHOD INTERNAL GetNumberOfSuccessfulTests : UINT
GetNumberOfSuccessfulTests := GetNumberOfTests() - GetNumberOfFailedTests() - GetNumberOfSkippedTests();
END_METHOD

METHOD INTERNAL GetNumberOfTests : UINT
GetNumberOfTests := NumberOfTests;
END_METHOD

METHOD INTERNAL GetNumberOfTestsToAnalyse : UINT
GetNumberOfTestsToAnalyse := MIN(GetNumberOfTests(), GVL_Param_TcUnit.MaxNumberOfTestsForEachTestSuite);
END_METHOD

METHOD GetTestByName : REFERENCE TO FB_Test
VAR_INPUT
  TestName : T_MaxString;
END_VAR
VAR
  IteratorCounter : UINT;
  NumberOfTestsToAnalyse : UINT(1..GVL_Param_TcUnit.MaxNumberOfTestSuites);
END_VAR
NumberOfTestsToAnalyse := GetNumberOfTestsToAnalyse();
FOR IteratorCounter := 1 TO NumberOfTestsToAnalyse BY 1 DO
  IF Tests[IteratorCounter].GetName() = TestName THEN
    GetTestByName REF= Tests[IteratorCounter];
    RETURN;
	END_IF
END_FOR
END_METHOD

// This method returns the test at the n'th position, ranging from 1.. NumberOfTests
METHOD INTERNAL GetTestByPosition : FB_Test
VAR_INPUT
    Position : UINT(1..GVL_Param_TcUnit.MaxNumberOfTestsForEachTestSuite);
END_VAR
GetTestByPosition := Tests[Position];
END_METHOD

METHOD INTERNAL GetTestOrderNumber : UINT(0..GVL_Param_TcUnit.MaxNumberOfTestsForEachTestSuite);
VAR_INPUT
    TestName : T_MaxString;
END_VAR
VAR
    IteratorCounter : UINT;
    NumberOfTestsToAnalyse : UINT(1..GVL_Param_TcUnit.MaxNumberOfTestsForEachTestSuite);
END_VAR
// Limit the test analyse to the max array limit of 'Tests[]'
NumberOfTestsToAnalyse := GetNumberOfTestsToAnalyse();

FOR IteratorCounter := 1 TO NumberOfTestsToAnalyse BY 1 DO
    IF Tests[IteratorCounter].GetName() = TestName THEN
        GetTestOrderNumber := Tests[IteratorCounter].GetTestOrder();
        RETURN;
    END_IF
END_FOR
END_METHOD

METHOD INTERNAL IsTestFinished : BOOL
VAR_INPUT
    TestName : T_MaxString;
END_VAR
VAR
    IteratorCounter : UINT;
    NumberOfTestsToAnalyse : UINT(0..GVL_Param_TcUnit.MaxNumberOfTestsForEachTestSuite);
END_VAR
// Limit the test analyse to the max array limit of 'Tests[]'
NumberOfTestsToAnalyse := GetNumberOfTestsToAnalyse();

IsTestFinished := FALSE;
FOR IteratorCounter := 1 TO NumberOfTestsToAnalyse BY 1 DO
    IF Tests[IteratorCounter].GetName() = TestName THEN
        IsTestFinished := Tests[IteratorCounter].IsFinished();
        RETURN;
    END_IF
END_FOR
END_METHOD

METHOD INTERNAL SetStartedAtIfNotSet
VAR_INPUT
    Timestamp : LWORD; // CPU cycle counter with 100ns precision
END_VAR
IF StartedAt = 0 THEN
    StartedAt := Timestamp;
END_IF
END_METHOD

METHOD INTERNAL SetStartedAtTimeBasedOnCpuCounter
StartedAt := F_GetCpuCounterAs64bit(GVL_TcUnit.GetCpuCounter);
END_METHOD

METHOD INTERNAL SetTestFailed
VAR_INPUT
    AssertionType : E_AssertionType;
    AssertionMessage : T_MaxString;
END_VAR
VAR
    IteratorCounter : UINT;
    NumberOfTestsToAnalyse : UINT(0..GVL_Param_TcUnit.MaxNumberOfTestsForEachTestSuite);
END_VAR
// Limit the test analyse to the max array limit of 'Tests[]'
NumberOfTestsToAnalyse := GetNumberOfTestsToAnalyse();

FOR IteratorCounter := 1 TO NumberOfTestsToAnalyse BY 1 DO
    IF Tests[IteratorCounter].GetName() = GVL_TcUnit.CurrentTestNameBeingCalled THEN
        Tests[IteratorCounter].SetFailed();
        Tests[IteratorCounter].SetAssertionType(AssertType := AssertionType);
        Tests[IteratorCounter].SetAssertionMessage(AssertMessage := AssertionMessage);
    END_IF
END_FOR
END_METHOD

(* Marks the test as finished in this testsuite.
   Returns TRUE if test was found, and FALSE if a test with this name was not found in this testsuite *)
METHOD INTERNAL SetTestFinished : BOOL;
VAR_INPUT
    TestName : T_MaxString;
    FinishedAt : LWORD;
END_VAR
VAR
    IteratorCounter : UINT;
    NumberOfTestsToAnalyse : UINT(0..GVL_Param_TcUnit.MaxNumberOfTestsForEachTestSuite);
END_VAR
// Limit the test analyse to the max array limit of 'Tests[]'
NumberOfTestsToAnalyse := GetNumberOfTestsToAnalyse();
FOR IteratorCounter := 1 TO NumberOfTestsToAnalyse BY 1 DO
    IF Tests[IteratorCounter].GetName() = TestName THEN
		IF NOT Tests[IteratorCounter].IsFinished() THEN
        	Tests[IteratorCounter].SetFinishedAndDuration(FinishedAt := FinishedAt);
			IF Tests[IteratorCounter].IsFailed() THEN
				TraceWithSeverity(
					Message := CONCAT(CONCAT('TEST FAILED: ', TestName),
							   CONCAT(' (', CONCAT(LREAL_TO_STRING(Tests[IteratorCounter].GetDuration()), 's)'))),
					Severity := Global.TcEventSeverity.Warning);
			ELSE
				TraceWithSeverity(
					Message := CONCAT(CONCAT('TEST PASSED: ', TestName),
							   CONCAT(' (', CONCAT(LREAL_TO_STRING(Tests[IteratorCounter].GetDuration()), 's)'))),
					Severity := Global.TcEventSeverity.Info);
			END_IF
		END_IF
		SetTestFinished := TRUE;
        RETURN;
    END_IF
END_FOR
SetTestFinished := FALSE;
END_METHOD

END_FUNCTION_BLOCK

// ---- POUs/FB_TimedTestSuite.TcPOU
FUNCTION_BLOCK FB_TimedTestSuite EXTENDS FB_TestSuite
VAR
    TimedTestStates      : ARRAY[1..GVL_Param_TcUnit.MaxNumberOfTestsForEachTestSuite] OF ST_TimedTestState;
    _nActiveTimedTestIdx : UINT;
    (* Task cycle in which _nActiveTimedTestIdx was set; a wait helper only accepts
       the context if it was set in the same cycle (guards cross-scan staleness) *)
    _nActiveTimedTestCycle : UDINT;
    // One-shot for the out-of-context wait Error trace (cyclic path - must not storm)
    bOutOfContextWaitTraced : BOOL;
END_VAR

METHOD PRIVATE _FindTestIndex : UINT
VAR_INPUT
    TestName : T_MaxString;
END_VAR
VAR
    i : UINT;
    nMax : UINT;
END_VAR
_FindTestIndex := 0;
nMax := GetNumberOfTestsToAnalyse();
FOR i := 1 TO nMax BY 1 DO
    IF Tests[i].GetName() = TestName THEN
        _FindTestIndex := i;
        RETURN;
    END_IF
END_FOR
END_METHOD

(* Returns the timed-test index for a wait-helper call, or 0 when the call is
   out of context. Valid context requires all three: an index was set, it was
   set in the current task cycle (TEST_TIMED* ran earlier in this scan and
   selected this test for body execution), and the framework's current test
   name still matches (defense against later TEST() calls in the same scan). *)
METHOD PRIVATE _GetActiveWaitContext : UINT
VAR
    idx : UINT;
END_VAR
_GetActiveWaitContext := 0;
idx := _nActiveTimedTestIdx;
IF idx = 0 THEN
    RETURN;
END_IF

GetCurrentTaskIndex();
IF _nActiveTimedTestCycle <> TwinCAT_SystemInfoVarList._TaskInfo[GetCurrentTaskIndex.index].CycleCount THEN
    RETURN;
END_IF

IF Tests[idx].GetName() <> GVL_TcUnit.CurrentTestNameBeingCalled THEN
    RETURN;
END_IF

_GetActiveWaitContext := idx;
END_METHOD

METHOD PUBLIC GetTimedTestResult : ST_TimedTestResult
VAR_INPUT
    TestName : T_MaxString;
END_VAR
VAR
    idx  : UINT;
    Test : REFERENCE TO FB_Test;
END_VAR
// Normalize the same way TEST(), TEST_ORDERED(), and TEST_TIMED() do
TestName := F_LTrim(in := F_RTrim(in := TestName));

idx := _FindTestIndex(TestName := TestName);
IF idx = 0 THEN
    RETURN;
END_IF

Test REF= Tests[idx];
IF NOT __ISVALIDREF(Test) THEN
    RETURN;
END_IF

GetTimedTestResult.TestName := Test.GetName();
GetTimedTestResult.bIsFailed := Test.IsFailed();
GetTimedTestResult.bIsSkipped := Test.IsSkipped();
GetTimedTestResult.bIsFinished := Test.IsFinished();
GetTimedTestResult.sFailureMessage := Test.GetAssertionMessage();
GetTimedTestResult.eFailureType := Test.GetAssertionType();
GetTimedTestResult.nNumberOfAsserts := Test.GetNumberOfAssertions();
GetTimedTestResult.lrDuration := Test.GetDuration();
GetTimedTestResult.stTimedState := TimedTestStates[idx];
END_METHOD

METHOD PUBLIC TEST_TIMED : BOOL
VAR_INPUT
    TestName       : T_MaxString;
    tSafetyTimeout : TIME;
END_VAR
VAR
    idx         : UINT;
    lrElapsed   : LREAL;
    lrTimeout   : LREAL;
    sMsg        : T_MaxString;
END_VAR
TEST_TIMED := FALSE;

// Step 1: Reset context
_nActiveTimedTestIdx := 0;

// Step 2: Trim name
TestName := F_LTrim(in := F_RTrim(in := TestName));

// Step 3: Register test via free function TEST()
TEST(TestName := TestName);

// Step 4: Check skip/ignore
IF GVL_TcUnit.IgnoreCurrentTest THEN
    RETURN;
END_IF

// Step 5: Find test index
idx := _FindTestIndex(TestName := TestName);
IF idx = 0 THEN
    RETURN;
END_IF

// Step 6: Check already finished
IF TimedTestStates[idx].bSafetyTimedOut OR IsTestFinished(TestName := TestName) THEN
    GVL_TcUnit.CurrentTestIsFinished := TRUE;
    RETURN;
END_IF

// Step 7: Initialize on first call
IF NOT TimedTestStates[idx].bInitialized THEN
    TimedTestStates[idx].nSafetyStartTime := F_GetCpuCounterAs64bit(GVL_TcUnit.GetCpuCounter);
    TimedTestStates[idx].tSafetyTimeout := tSafetyTimeout;
    TimedTestStates[idx].bInitialized := TRUE;
END_IF

// Step 8: Check safety timeout (compare against stored value)
lrElapsed := ULINT_TO_LREAL(F_GetCpuCounterAs64bit(GVL_TcUnit.GetCpuCounter) - TimedTestStates[idx].nSafetyStartTime)
             * GVL_TcUnit.HundredNanosecondToSecond;
lrTimeout := TIME_TO_LREAL(TimedTestStates[idx].tSafetyTimeout) / 1000.0;

IF lrElapsed > lrTimeout THEN
    sMsg := CONCAT('SAFETY TIMEOUT: Test "', CONCAT(TestName, CONCAT('" exceeded ', LREAL_TO_FMTSTR(lrTimeout, 1, TRUE))));
    sMsg := CONCAT(sMsg, 's');

    SetTestFailed(AssertionType := E_AssertionType.Type_TIMEOUT,
                  AssertionMessage := sMsg);
    SetTestFinished(TestName := TestName,
                    FinishedAt := F_GetCpuCounterAs64bit(GVL_TcUnit.GetCpuCounter));
    CalculateAndSetNumberOfAssertsForTest(TestName := TestName);

    TimedTestStates[idx].bSafetyTimedOut := TRUE;
    GVL_TcUnit.CurrentTestIsFinished := TRUE;

    TraceWithSeverity(Message := sMsg, Severity := TcEventSeverity.Warning);
    RETURN;
END_IF

// Step 9: Test body should execute - arm the wait context for this cycle only
_nActiveTimedTestIdx := idx;
GetCurrentTaskIndex();
_nActiveTimedTestCycle := TwinCAT_SystemInfoVarList._TaskInfo[GetCurrentTaskIndex.index].CycleCount;
TEST_TIMED := TRUE;
END_METHOD

METHOD PUBLIC TEST_TIMED_ORDERED : BOOL
VAR_INPUT
    TestName       : T_MaxString;
    tSafetyTimeout : TIME;
END_VAR
VAR
    CounterTestSuiteAddress : UINT;
    SuiteIndex              : UINT;
    Test                    : REFERENCE TO FB_Test;
    idx                     : UINT;
    lrElapsed               : LREAL;
    lrTimeout               : LREAL;
    sMsg                    : T_MaxString;
END_VAR
TEST_TIMED_ORDERED := FALSE;

// Step 1: Reset context
_nActiveTimedTestIdx := 0;

// Step 2: Trim name (matches TEST_ORDERED line 34)
TestName := F_LTrim(in := F_RTrim(in := TestName));

// Step 3: Set global test name (matches line 37)
GVL_TcUnit.CurrentTestNameBeingCalled := TestName;

// Step 4: Find suite in runner registry (matches lines 44-47)
SuiteIndex := 0;
FOR CounterTestSuiteAddress := 1 TO GVL_TcUnit.NumberOfInitializedTestSuites BY 1 DO
    IF GVL_TcUnit.TestSuiteAddresses[CounterTestSuiteAddress] = GVL_TcUnit.CurrentTestSuiteBeingCalled THEN
        SuiteIndex := CounterTestSuiteAddress;
        EXIT;
    END_IF
END_FOR
IF SuiteIndex = 0 THEN
    RETURN;
END_IF

// Step 5: Register as ordered test (matches line 48)
Test REF= GVL_TcUnit.TestSuiteAddresses[SuiteIndex]^.AddTest(TestName := TestName, IsTestOrdered := TRUE);

// Step 6: Set CurrentTestIsFinished (matches line 49)
GVL_TcUnit.CurrentTestIsFinished := GVL_TcUnit.TestSuiteAddresses[SuiteIndex]^.IsTestFinished(TestName := TestName);

// Step 7: Check skip/ignore (matches lines 76-78)
IF GVL_TcUnit.IgnoreCurrentTest THEN
    RETURN;
END_IF

// Step 8: Check ordered cursor (matches lines 55-74)
IF GetTestOrderNumber(TestName := TestName) = GVL_TcUnit.CurrentlyRunningOrderedTestInTestSuite[SuiteIndex] THEN
    IF GVL_TcUnit.CurrentTestIsFinished THEN
        // Already finished - advance cursor (matches lines 58-62)
        GVL_TcUnit.CurrentlyRunningOrderedTestInTestSuite[SuiteIndex] :=
            GVL_TcUnit.CurrentlyRunningOrderedTestInTestSuite[SuiteIndex] + 1;
        GVL_TcUnit.IgnoreCurrentTest := TRUE;
        RETURN;
    END_IF
ELSE
    // Not this test's turn (matches lines 70-73)
    GVL_TcUnit.IgnoreCurrentTest := TRUE;
    RETURN;
END_IF

// --- From here: this test's turn AND not finished. Add timed-test logic. ---

// Step 9: Find timed test index
idx := _FindTestIndex(TestName := TestName);
IF idx = 0 THEN
    RETURN;
END_IF

// Step 10: Check already timed out
IF TimedTestStates[idx].bSafetyTimedOut THEN
    GVL_TcUnit.CurrentTestIsFinished := TRUE;
    RETURN;
END_IF

// Step 11: Initialize on first call
IF NOT TimedTestStates[idx].bInitialized THEN
    TimedTestStates[idx].nSafetyStartTime := F_GetCpuCounterAs64bit(GVL_TcUnit.GetCpuCounter);
    TimedTestStates[idx].tSafetyTimeout := tSafetyTimeout;
    TimedTestStates[idx].bInitialized := TRUE;
END_IF

// Step 12: Check safety timeout (compare against stored value)
lrElapsed := ULINT_TO_LREAL(F_GetCpuCounterAs64bit(GVL_TcUnit.GetCpuCounter) - TimedTestStates[idx].nSafetyStartTime)
             * GVL_TcUnit.HundredNanosecondToSecond;
lrTimeout := TIME_TO_LREAL(TimedTestStates[idx].tSafetyTimeout) / 1000.0;

IF lrElapsed > lrTimeout THEN
    sMsg := CONCAT('SAFETY TIMEOUT: Test "', CONCAT(TestName, CONCAT('" exceeded ', LREAL_TO_FMTSTR(lrTimeout, 1, TRUE))));
    sMsg := CONCAT(sMsg, 's');

    SetTestFailed(AssertionType := E_AssertionType.Type_TIMEOUT,
                  AssertionMessage := sMsg);
    SetTestFinished(TestName := TestName,
                    FinishedAt := F_GetCpuCounterAs64bit(GVL_TcUnit.GetCpuCounter));
    CalculateAndSetNumberOfAssertsForTest(TestName := TestName);

    TimedTestStates[idx].bSafetyTimedOut := TRUE;
    GVL_TcUnit.CurrentTestIsFinished := TRUE;

    TraceWithSeverity(Message := sMsg, Severity := TcEventSeverity.Warning);
    RETURN;
END_IF

// Step 13: Set started timestamp (matches line 66)
IF __ISVALIDREF(Test) THEN
    Test.SetStartedAtIfNotSet(Timestamp := F_GetCpuCounterAs64bit(GVL_TcUnit.GetCpuCounter));
END_IF

// Step 14: Test body should execute - arm the wait context for this cycle only
_nActiveTimedTestIdx := idx;
GetCurrentTaskIndex();
_nActiveTimedTestCycle := TwinCAT_SystemInfoVarList._TaskInfo[GetCurrentTaskIndex.index].CycleCount;
TEST_TIMED_ORDERED := TRUE;
END_METHOD

METHOD PUBLIC WaitForCondition : BOOL
VAR_INPUT
    bCondition : BOOL;
    tTimeout   : TIME;
END_VAR
VAR
    idx       : UINT;
    lrElapsed : LREAL;
    lrTarget  : LREAL;
END_VAR
WaitForCondition := FALSE;
idx := _GetActiveWaitContext();

// Step 1: Context check (one-shot trace - this path is cyclic)
IF idx = 0 THEN
    IF NOT bOutOfContextWaitTraced THEN
        bOutOfContextWaitTraced := TRUE;
        TraceWithSeverity(
            Message := 'WaitForCondition called without active timed test context',
            Severity := TcEventSeverity.Error);
    END_IF
    RETURN;
END_IF

// Step 2: Pass-through if already complete
IF TimedTestStates[idx].bWaitComplete THEN
    WaitForCondition := TRUE;
    RETURN;
END_IF

// Step 3: Type mismatch check
IF TimedTestStates[idx].eWaitType = E_WaitType.Duration THEN
    SetTestFailed(AssertionType := E_AssertionType.Type_WAIT_MISUSE,
                  AssertionMessage := 'WaitForCondition called but WaitForTime already active');
    SetTestFinished(TestName := GVL_TcUnit.CurrentTestNameBeingCalled,
                    FinishedAt := F_GetCpuCounterAs64bit(GVL_TcUnit.GetCpuCounter));
    CalculateAndSetNumberOfAssertsForTest(TestName := GVL_TcUnit.CurrentTestNameBeingCalled);
    GVL_TcUnit.CurrentTestIsFinished := TRUE;
    RETURN;
END_IF

// Step 4: First call with condition already TRUE - immediate completion
IF bCondition AND TimedTestStates[idx].nWaitStartTime = 0 THEN
    TimedTestStates[idx].bWaitComplete := TRUE;
    TimedTestStates[idx].bConditionTimedOut := FALSE;
    TimedTestStates[idx].eWaitType := E_WaitType.Condition;
    TraceWithSeverity(
        Message := CONCAT('WaitForCondition: condition already TRUE for test "', CONCAT(GVL_TcUnit.CurrentTestNameBeingCalled, '"')),
        Severity := TcEventSeverity.Info);
    WaitForCondition := TRUE;
    RETURN;
END_IF

// Step 5: First call, condition not yet met - start wait
IF TimedTestStates[idx].nWaitStartTime = 0 THEN
    TimedTestStates[idx].eWaitType := E_WaitType.Condition;
    TimedTestStates[idx].tLatchedDuration := tTimeout;
    TimedTestStates[idx].nWaitStartTime := F_GetCpuCounterAs64bit(GVL_TcUnit.GetCpuCounter);
    TraceWithSeverity(
        Message := CONCAT('WaitForCondition started: timeout ', CONCAT(TIME_TO_STRING(tTimeout), CONCAT(' for test "', CONCAT(GVL_TcUnit.CurrentTestNameBeingCalled, '"')))),
        Severity := TcEventSeverity.Verbose);
    RETURN;
END_IF

// Step 6: Condition met during wait
IF bCondition THEN
    TimedTestStates[idx].bWaitComplete := TRUE;
    TimedTestStates[idx].bConditionTimedOut := FALSE;
    TraceWithSeverity(
        Message := CONCAT('WaitForCondition: condition met for test "', CONCAT(GVL_TcUnit.CurrentTestNameBeingCalled, '"')),
        Severity := TcEventSeverity.Info);
    WaitForCondition := TRUE;
    RETURN;
END_IF

// Step 7: Check timeout
lrElapsed := ULINT_TO_LREAL(F_GetCpuCounterAs64bit(GVL_TcUnit.GetCpuCounter) - TimedTestStates[idx].nWaitStartTime)
             * GVL_TcUnit.HundredNanosecondToSecond;
lrTarget := TIME_TO_LREAL(TimedTestStates[idx].tLatchedDuration) / 1000.0;

IF lrElapsed >= lrTarget THEN
    TimedTestStates[idx].bWaitComplete := TRUE;
    TimedTestStates[idx].bConditionTimedOut := TRUE;
    TraceWithSeverity(
        Message := CONCAT('WaitForCondition timed out after ', CONCAT(LREAL_TO_FMTSTR(lrElapsed, 3, TRUE), CONCAT('s for test "', CONCAT(GVL_TcUnit.CurrentTestNameBeingCalled, '"')))),
        Severity := TcEventSeverity.Warning);
    WaitForCondition := TRUE;
END_IF

// Step 8: Still waiting - return FALSE (default)
END_METHOD

METHOD PUBLIC WaitForTime : BOOL
VAR_INPUT
    tDuration : TIME;
END_VAR
VAR
    idx       : UINT;
    lrElapsed : LREAL;
    lrTarget  : LREAL;
END_VAR
WaitForTime := FALSE;
idx := _GetActiveWaitContext();

// Step 1: Context check (one-shot trace - this path is cyclic)
IF idx = 0 THEN
    IF NOT bOutOfContextWaitTraced THEN
        bOutOfContextWaitTraced := TRUE;
        TraceWithSeverity(
            Message := 'WaitForTime called without active timed test context',
            Severity := TcEventSeverity.Error);
    END_IF
    RETURN;
END_IF

// Step 2: Pass-through if already complete
IF TimedTestStates[idx].bWaitComplete THEN
    WaitForTime := TRUE;
    RETURN;
END_IF

// Step 3: Type mismatch check
IF TimedTestStates[idx].eWaitType = E_WaitType.Condition THEN
    SetTestFailed(AssertionType := E_AssertionType.Type_WAIT_MISUSE,
                  AssertionMessage := 'WaitForTime called but WaitForCondition already active');
    SetTestFinished(TestName := GVL_TcUnit.CurrentTestNameBeingCalled,
                    FinishedAt := F_GetCpuCounterAs64bit(GVL_TcUnit.GetCpuCounter));
    CalculateAndSetNumberOfAssertsForTest(TestName := GVL_TcUnit.CurrentTestNameBeingCalled);
    GVL_TcUnit.CurrentTestIsFinished := TRUE;
    RETURN;
END_IF

// Step 4: First call - start wait
IF TimedTestStates[idx].nWaitStartTime = 0 THEN
    TimedTestStates[idx].eWaitType := E_WaitType.Duration;
    TimedTestStates[idx].tLatchedDuration := tDuration;
    TimedTestStates[idx].nWaitStartTime := F_GetCpuCounterAs64bit(GVL_TcUnit.GetCpuCounter);
    TraceWithSeverity(
        Message := CONCAT('Wait started: ', CONCAT(TIME_TO_STRING(tDuration), CONCAT(' for test "', CONCAT(GVL_TcUnit.CurrentTestNameBeingCalled, '"')))),
        Severity := TcEventSeverity.Verbose);
    RETURN;
END_IF

// Steps 5-8: Check elapsed
lrElapsed := ULINT_TO_LREAL(F_GetCpuCounterAs64bit(GVL_TcUnit.GetCpuCounter) - TimedTestStates[idx].nWaitStartTime)
             * GVL_TcUnit.HundredNanosecondToSecond;
lrTarget := TIME_TO_LREAL(TimedTestStates[idx].tLatchedDuration) / 1000.0;

IF lrElapsed >= lrTarget THEN
    TimedTestStates[idx].bWaitComplete := TRUE;
    TraceWithSeverity(
        Message := CONCAT('Wait completed: ', CONCAT(LREAL_TO_FMTSTR(lrElapsed, 3, TRUE), CONCAT('s elapsed for test "', CONCAT(GVL_TcUnit.CurrentTestNameBeingCalled, '"')))),
        Severity := TcEventSeverity.Info);
    WaitForTime := TRUE;
END_IF
END_METHOD

PROPERTY PUBLIC WaitTimedOut : BOOL
GET
VAR
    idx : UINT;
END_VAR
idx := _GetActiveWaitContext();
IF idx > 0 THEN
    WaitTimedOut := TimedTestStates[idx].bConditionTimedOut;
ELSE
    WaitTimedOut := FALSE;
END_IF
END_GET
END_PROPERTY

END_FUNCTION_BLOCK
